// TIA Portal V20 export
FUNCTION_BLOCK "progalarme"   // FB3, LAD
{ S7_Optimized_Access := 'TRUE' }
// stored: MemoryReserve 100, SetENOAutomatically false
   VAR_INPUT
      AlarmInput : Bool;
      AlarmText : String;
      Tag : String;
   END_VAR
   VAR_IN_OUT
      Program_Alarm_1 : Program_Alarm;
   END_VAR
   VAR
      Program_Alarm_2 { S7_SetPoint := 'True'} : Program_Alarm;
   END_VAR
   VAR_TEMP
      Error : Bool;
      Status : Word;
   END_VAR
BEGIN

REGION Network 1
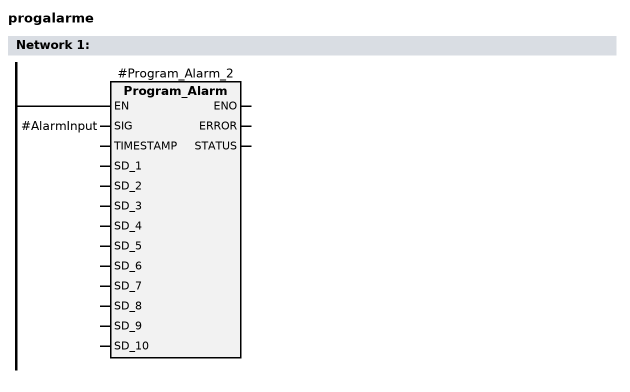
   RUNG wire#powerrail
      #Program_Alarm_2.Program_Alarm(SIG := #AlarmInput, TIMESTAMP :=, SD_1 :=, SD_2 :=, SD_3 :=, SD_4 :=, SD_5 :=, SD_6 :=, SD_7 :=, SD_8 :=, SD_9 :=, SD_10 :=, Error =>, Status =>)
   END_RUNG
   // the same network as SCL:
   #Program_Alarm_2(SIG := #AlarmInput);   // Program_Alarm
END_REGION
END_FUNCTION_BLOCK
